{attribute 'GeneratedUsingTerminal: EJ9505-0000-0016'}
{attribute addProperty BoxType "EJ9505-0000-0016"}
{attribute addProperty Id "Power_OKAT %I*BOOL1OverloadAT %I*BOOL1"}
{attribute addProperty CRC "3101291258"}
{attribute addProperty Size "2"}
TYPE Status_Uo_B8D9F2FA EXTENDS InputBase_8311D824 :
STRUCT
	{attribute addProperty Name "Power_OK"}
	Power_OK AT %I* : BOOL;
	{attribute addProperty Name "Overload"}
	Overload AT %I* : BOOL;
END_STRUCT
END_TYPE

(* stored: Version 1.2.0.0, ProductVersion 3.1.4024.9
   DUT Status_Uo_B8D9F2FA: Id {878e15f9-cb20-4694-a459-c85049c367ee} *)
